PROGRAM MAIN
VAR
	bFirstCycle : BOOL := TRUE;
	Boiler : FB_Boiler;
	
	TempChange : LREAL;
	lastTemp : LREAL;
END_VAR

IF bFirstCycle THEN
	Boiler.SimulateComponents := TRUE;
END_IF

Boiler.CyclicLogic();

TempChange := Boiler.CurrentTemp - lastTemp;
lastTemp := Boiler.CurrentTemp;
;

END_PROGRAM

(* stored: Version 1.1.0.1
   POU MAIN: Id {5476d895-76ae-435d-9782-f6b13de03fcd}, SpecialFunc None *)
